// TIA Portal V20 export
VAR_GLOBAL   // PLC tag table "LPFE_Constants"
END_VAR
VAR_GLOBAL CONSTANT   // user constants
   MAX_NO_PROGRAMS : UInt := 20;   // Maximum Number of configured Programs
   BYTE_ARRAY_LENGTH_WO_HEADER_OUT : UDInt := 944;   // Array size without Header Outgoing Message
   INBOUND_TIMEOUT : Time := T#10s;   // Time until hasTimeout becomes true when seq and ack differ
   DINT_ARRAY_LENGTH : Int := 99;   // Upper bound of DINT Array. Array real size is this value+1
   NUMBER_MESSAGES_PRT_BUFFER : Int := 100;   // Number of messages contained in PR&T Buffer
   TIMEOUT_INTERVAL : Time := T#10s;   // Interval configured to receive the acknowledge message of an event before starting the retry sequence
   LE_NUMBER_OF_INTERFACE_BUFFERS : Int := 2;   // Upper bound of 'toHost' Channels Array. Array real size is this value+1
   LE_NUMBER_MESSAGES_ACK_BUFFER : Int := 9;   // Upper bound of AcknowledgeBuffer. Array real size is this value+1
   RETRY_ON_TIME : Time := T#2s;   // Interval where the retry sequence starts
   NO_OF_CELLS : UInt := 4;   // Number of configured Cells
   NUMBER_TXN_PER_MESSAGE : Int := 9;   // Upper bound of txnBuffer Array. Array real size is this value+1
   NUMBER_MESSAGES_ACK_BUFFER : Int := 10;   // Number of messages contained in Acknowledge Buffer
   LE_NUMBER_MESSAGES_RECORD_BUFFER : Int := 99;   // Upper bound of RecordBuffer. Array real size is this value+1
   NUMBER_MESSAGES_RECORD_BUFFER : Int := 100;   // Number of messages contained in Record Buffer
   BYTE_ARRAY_LENGTH : Int := 999;   // Upper bound of Message Byte Array. Array real size is this value+1
   LE_NUMBER_MSGS_PER_INTERFACE_BUFFER : Int := 1;   // Upper bound of 'toHost' Buffer Array. Array real size is this value+1
   RETRY_INTERVAL : Time := T#10s;   // Interval to trigger a new retry message after the retry sequence started
   CONFIGURED_ALARMS : UInt := 999;   // Upper Bound of Additional Alarm Data Array . Array real size is this value+1
   BYTE_ARRAY_LENGTH_WO_HEADER_IN : UDInt := 376;   // Array size without Header Incoming Message
   NUMBER_MSGS_PER_INTERFACE_BUFFER : Int := 2;   // Buffer size of the in and out data channels
   SIZE_TRANSACTIONS_ARRAY : Int := 9;   // Upper bound of Monitor Transactions Array. Array real size is this value+1
   LE_NUMBER_MESSAGES_PRT_BUFFER : Int := 99;   // Upper bound of PRTBuffer. Array real size is this value+1
   LE_NUMBER_MESSAGES_MAIN_BUFFER : Int := 49;   // Upper bound of Main Buffer. Array real size is this value+1
   NUMBER_MESSAGES_MAIN_BUFFER : Int := 50;   // Number of messages contained in Main Buffer
   LE_NUMBER_MESSAGES_FN_BUFFER : Int := 19;   // Upper bound of FlexNetBuffer. Array real size is this value+1
   NUMBER_MESSAGES_FN_BUFFER : Int := 20;   // Number of messages contained in FlexNet Buffer
   LE_NUMBER_MESSAGES_TELEMETRY_BUFFER : Int := 19;   // Upper bound of TelemetryBuffer. Array real size is this value+1
   NUMBER_MESSAGES_TELEMETRY_BUFFER : Int := 20;   // Number of messages contained in Telemetry Buffer
END_VAR
